TEXTLIST TL_RecipesManagerStatus_1
  0 = 'Idle'
  10 = 'Initialization'
  20 = 'Create'
  30 = 'Load'
  40 = 'Read'
  50 = 'Reload'
  60 = 'Backup'
  70 = 'Restore'
  -10 = 'Abort'
   = ''
END_TEXTLIST

(* stored: Version 1.1.0.1, ProductVersion 3.1.4024.12
   TextList TL_RecipesManagerStatus_1: Id {91297877-3e68-45d3-a09a-142f45db2d48} *)
